Fanuc TP program (LS listing): at_place.ls

/PROG  AT_PLACE
/ATTR
COMMENT		= "";
DEFAULT_GROUP	= 1,*,*,*,*;
/MN
 : UFRAME_NUM=2 ;
 : UTOOL_NUM=2 ;
 : PR[2:LPOS]=LPOS ;
 : IF (PR[2,1]<(-100)),JMP LBL[500] ;
 : IF (PR[2,1]<100),JMP LBL[500] ;
 : IF (PR[2,2]<(-100)),JMP LBL[500] ;
 : IF (PR[2,2]<100),JMP LBL[500] ;
 : IF (PR[2,3]<(-100)),JMP LBL[500] ;
 : IF (PR[2,3]<(-100)),JMP LBL[500] ;
 : R[2:zoneID]=2 ;
 : END ;
 :  ;
 : LBL[500] ;
 :   R[2:zoneID]=0 ;
 :   END ;
/POS
/END
